(* Logix 5000 project; controller cal1615 1756-L62 rev 20.19; software revision 20.05; part 2 of 82 *)

TYPE Accumulator :
STRUCT
   OUT_Not_EStop : BOOL;   // E-Stop Not Requested
   OUT_Not_Fast_Stop : BOOL;   // Fast Stop Not Requested
   OUT_Not_Normal_Stop : BOOL;   // Normal Stop Not Requested
   OUT_Request_Line_Slowdown : BOOL;   // Request Line Slowdown
   OUT_Full : BOOL;   // Accumulator is Full
   OUT_Empty : BOOL;   // Accumulator is Empty
   OUT_Alarm : BOOL;   // Alarm Exists
   OUT_Unack_Alarm : BOOL;   // Unacknowledged Alarm Exists
   OUT_Warning : BOOL;   // Warning Exists
   OUT_Unack_Warning : BOOL;   // Unacknowledged Warning Exists
   OUT_control_limit : BOOL;   // Control Limit Position
   OUT_Speed : REAL;   // Output Speed
   OUT_Nip_Close : BOOL;   // Nip Close Request
   IN_Speed : REAL;   // Input Speed
   OUT_Acc_Payout : BOOL;   // Accumulator Payout
   OUT_Close_Nip : BOOL;   // Close Nip
   OUT_Acc_Fill_Request : BOOL;   // Accumulator Fill Request
END_STRUCT
END_TYPE

TYPE acs800_di_normal :
STRUCT
   faulted : BOOL;
   warning : BOOL;
   running_fwd : BOOL;
   running_rev : BOOL;
   ready : BOOL;
   ctrl_from_net : BOOL;
   ref_from_net : BOOL;
   at_reference : BOOL;
END_STRUCT
END_TYPE

TYPE acs800_do_normal :
STRUCT
   forward : BOOL;
   reverse : BOOL;
   fault_reset : BOOL;
   net_control : BOOL;
   net_reference : BOOL;
END_STRUCT
END_TYPE

TYPE hmi_dint :
STRUCT
   hmi : DINT[16];
   global : DINT[16];
   zone_1 : DINT[16];
   zone_2 : DINT[16];
   zone_3 : DINT[16];
   letoff : DINT[16];
   ts1 : DINT[16];
   ts2 : DINT[16];
   upl : DINT[16];
   lpl : DINT[16];
   wdr : DINT[16];
   wdt : DINT[16];
   splice : DINT[16];
   mrc : DINT[16];
   static : DINT[16];
   imp : DINT[16];
   misc : DINT[16];
   edg : DINT[16];
   slt : DINT[16];
   impreg : DINT[16];
   adv_cooling : DINT[16];
   retraction : DINT[16];
END_STRUCT
END_TYPE

TYPE hmi_real :
STRUCT
   hmi : REAL[112];
   global : REAL[112];
   zone_1 : REAL[112];
   zone_2 : REAL[112];
   zone_3 : REAL[112];
   letoff : REAL[112];
   ts1 : REAL[112];
   ts2 : REAL[112];
   upl : REAL[112];
   lpl : REAL[112];
   wdr : REAL[112];
   wdt : REAL[112];
   splice : REAL[112];
   mrc : REAL[112];
   static : REAL[112];
   impreg : REAL[112];
   misc : REAL[112];
   edg : REAL[112];
   slt : REAL[112];
   adv_cooling : REAL[112];
END_STRUCT
END_TYPE

TYPE PIDE :   // PIDE
STRUCT
   pide_ctrl : PID_ENHANCED;   // Control PID
   pide_autotune : PIDE_AUTOTUNE;   // PID Autotune Data
   ao_cv : REAL;   // Analog Output: Temperature Control Valve
   param_cv_min : REAL;   // Control Valve Minimum Output
   param_cv_max : REAL;   // Control Valve Maximum Output
   param_pv_min : REAL;   // PV Minimum
   param_pv_max : REAL;   // PV Maximum
   pid_manual_sp : REAL;   // Manual Mode Control Valve Setpoint
   pid_ctrl_cv : REAL;   // Control Valve Output
   pid_ctrl_pv : REAL;   // Control Process Variable
   pid_ctrl_sp : REAL;   // Control Setpoint
   pid_ctrl_sp_error : REAL;   // Control Absolute Error
   pid_ctrl_sp_last : REAL;   // Control Setpoint Last Scan
   oneshot : DINT;   // One Shot
   status : DINT;   // Run Status
   enable_deviation_alarm : BOOL;   // Enable Temperature Deviation Alarm
   pb_cv_manual : BOOL;   // Manual Mode Pushbutton
   pb_cv_auto : BOOL;   // Auto Mode Pushbutton
   pid_manual_mode : BOOL;   // Manual Mode
   request_pid_control : BOOL;   // PID Control Request
   request_manual : BOOL;   // PID Manual Mode Request
END_STRUCT
END_TYPE

TYPE recipe :
STRUCT
   name : STRING;
   comments : STRING;
   master_line_speed : REAL;
   zone_1 : zone;
   zone_2 : zone;
   zone_3 : zone;
   line_speed_sp : REAL;
   letoff_tension_sp : REAL;
   acc_tension_sp : REAL;
   acc_fill_pressure_sp : REAL;
   acc_counter_pressure_sp : REAL;
   cure_time_sp : REAL;
   platen_temp_sp : REAL;
   impreg_gap_sp : REAL;
   impreg_gap_ds_offset_sp : REAL;
   impreg_gap_os_offset_sp : REAL;
   impreg_supply_speed_sp : REAL;
   impreg_roll_speed_sp : REAL;
   ts1_mode_sp : REAL;
   ts1_tension_sp : REAL;
   ts1_stretch_sp : REAL;
   liner_winder_brake_sp : REAL;
   slitter_speed_sp : REAL;
   adv_cooling_temp_sp : REAL;
   ts2_tension_sp : REAL;
   lower_poly_tension_sp : REAL;
   lower_poly_b_tension_sp : REAL;
   upper_poly_tension_sp : REAL;
   upper_poly_b_tension_sp : REAL;
   winder_tension_sp : REAL;
   winder_mode_sp : REAL;
   winder_torque_sp : REAL;
   tension_deviation_sp : REAL;
   winder_tension_sp_max : REAL;
   winder_tension_sp_min : REAL;
END_STRUCT
END_TYPE

TYPE routine :
STRUCT
   comment : DINT;
   oneshot : DINT;
   fault : DINT;
   fault_ack : DINT;
   fault1 : DINT;
   fault1_ack : DINT;
   warning : DINT;
   warning_ack : DINT;
   unack_fault : BOOL;
   unack_warning : BOOL;
   state : DINT;
END_STRUCT
END_TYPE

TYPE servo_di :
STRUCT
   mode_bit_0 : BOOL;
   mode_bit_1 : BOOL;
   homed : BOOL;
   stand_still : BOOL;
   at_target_pos : BOOL;
   command_change : BOOL;
   operator_mode_error : BOOL;
   drive_does_not_follow : BOOL;
   actual_op_mode_bit_0 : BOOL;
   actual_op_mode_bit_1 : BOOL;
   class_3_diagnostic : BOOL;
   class_2_diagnostic : BOOL;
   class_1_diagnostic : BOOL;
   operation_bit_14 : BOOL;
   operation_bit_15 : BOOL;
END_STRUCT
END_TYPE

TYPE servo_do :
STRUCT
   command_value_accept : BOOL;
   fault_reset : BOOL;
   jog_forward : BOOL;
   jog_reverse : BOOL;
   jog_enable : BOOL;
   drive_halt_0_halt : BOOL;
   drive_enable : BOOL;
   ready_for_operation_bit_16 : BOOL;
   ready_for_operation_bit_17 : BOOL;
END_STRUCT
END_TYPE

TYPE Setpoint :   // ******************** DO NOT CHANGE ORDER OF TAGS ******************** ****
STRUCT
   SP : REAL;   // Setpoint
   Lo : REAL;   // Lo
   Hi : REAL;   // Hi
END_STRUCT
END_TYPE

TYPE vfd_data :
STRUCT
   In_OutputFreq : DINT;
   In_RPM : DINT;
   In_OutputCurrent : DINT;
   In_MaximumFreq : DINT;
   In_MotorNPHz : DINT;
   In_MotorNPRPM : DINT;
   In_DriveStatus : DINT;
   Out_CommandedFreq : DINT;
   Out_DriveLogicRslt : DINT;
   Out_CommandedRPM : DINT;
   In_DriveStatus_Ready : BOOL;
   In_DriveStatus_Active : BOOL;
   In_DriveStatus_Faulted : BOOL;
   In_DriveStatus_Net : BOOL;
   In_DriveStatus_AtReference : BOOL;
   Out_DriveLogicRslt_Stop : BOOL;
   Out_DriveLogicRslt_Start : BOOL;
   Out_DriveLogicRslt_ClearFault : BOOL;
   Out_DriveLogicRslt_Forward : BOOL;
   Out_DriveLogicRslt_Reverse : BOOL;
END_STRUCT
END_TYPE

TYPE vfd_data_ACS880 :
STRUCT
   In_OutputRPM : DINT;   // Input
   In_OutputCurrent : DINT;   // Input
   IN_OutputHz : DINT;   // Output Hz
   IN_OutputTorque : DINT;   // Input Motor Torque
   In_SpeedScaling : DINT;   // Input
   In_MotorNPHz : DINT;   // Input
   In_MotorNPRPM : DINT;   // Input
   In_DriveStatus : DINT;   // Input
   Out_DriveLogicRslt : DINT;   // Output
   Out_Speed_Setpoint : REAL;   // Motor Speed Setpoint in Engineering Units
   Out_SpeedScaling : DINT;   // Output Speed Scaling
   Out_Commanded_SPEED : REAL;   // Output
   Out_Commanded_Torque : REAL;   // Output Torque
   C_speed_hz : BOOL;   // Speed Setpoint in Hz
   C_speed_pct : BOOL;   // Speed Setpoint In Percent
   C_speed_rpm : BOOL;   // Speed Setpoint in RPM
   In_DriveStatus_RDY_ON : BOOL;   // Input
   In_DriveStatus_RDY_RUN : BOOL;   // Input
   In_DriveStatus_RDY_REF : BOOL;   // Input
   In_DriveStatus_TRIPPED : BOOL;   // Input Status Tripped
   In_DriveStatus_OFF_2_STA : BOOL;   // Input Status Off 2 State
   In_DriveStatus_OFF_3_STA : BOOL;   // Input Status Off 3 State
   In_DriveStatus_SWC_ON_INHIB : BOOL;   // Input Status SWC On Inhibit
   In_DriveStatus_ALARM : BOOL;   // Input Status Alarm
   In_DriveStatus_AT_SETPOINT : BOOL;   // Input Status At Setpoint
   In_DriveStatus_REMOTE : BOOL;   // Input Status Remote
   In_DriveStatus_ABOVE_LIMIT : BOOL;   // Input Status Above Limit
   In_DriveStatus_EXT_CTRL_LOC : BOOL;   // Input Status External Control
   In_DriveStatus_EXT_RUN_ENABLE : BOOL;   // Input Status External Run Enable
   In_DriveStatus_FBA_ERROR : BOOL;   // Input Status Field Bus Error
   Out_DriveLogicRslt_OFF1_CONTROL : BOOL;   // Output Off 1 Control
   Out_DriveLogicRslt_OFF2_CONTROL : BOOL;   // Output Off 2 Control
   Out_DriveLogicRslt_OFF3_CONTROL : BOOL;   // Output Off 3 Control
   Out_DriveLogicRslt_INHIBIT_OPERATION : BOOL;   // Output Inhibit Operation
   Out_DriveLogicRslt_RAMP_OUT_ZERO : BOOL;   // Output Ramp Out Zero
   Out_DriveLogicRslt_RAMP_HOLD : BOOL;   // Output Ramp Hold
   Out_DriveLogicRslt_RAMP_IN_ZERO : BOOL;   // Output Ramp In Zero
   Out_DriveLogicRslt_RESET : BOOL;   // Output Reset
   Out_DriveLogicRslt_REMOTE_CMD : BOOL;   // Output Remmote Command
   Out_DriveLogicRslt_EXT_CTRL_LOC : BOOL;   // Output Ext Ctrl Loc
   OUT_Comm_Status : BOOL;
END_STRUCT
END_TYPE

TYPE zone :
STRUCT
   recirc_sp : REAL;
   exhaust_sp : REAL;
   temp_sp : REAL;
END_STRUCT
END_TYPE

ADD_ON_INSTRUCTION ABB_PROTOCOL_VFD   (* revision 1.0 *)
VAR_INPUT
   STATUS_WORD : INT; {required}
END_VAR
VAR_OUTPUT
   CONTROL_WORD : INT; {access Read Only, required}
END_VAR
VAR_INPUT
   DRIVE_NOT_READY_FAULT : BOOL;
END_VAR
VAR_OUTPUT
   OUT_FAULT : BOOL; {access Read Only, visible}
   OUT_ALARM : BOOL; {access Read Only, visible}
   OUT_ENABLED : BOOL; {access Read Only, visible}
END_VAR
VAR_INPUT
   IN_START : BOOL; {required}
   IN_GLOBAL_RESET : BOOL; {required}
   IN_DRIVE_PERMISSIVE : BOOL; {required}
END_VAR
VAR
   run_permissive : BOOL;
   enable_drives : BOOL;
   request_run : BOOL;
   drive_on_request : BOOL;
   seq : routine;
   step_3_timer : TIMER := (PRE := 500);
   fault_timer : TIMER := (PRE := 2000);
END_VAR

ROUTINE Logic   (* ladder *)
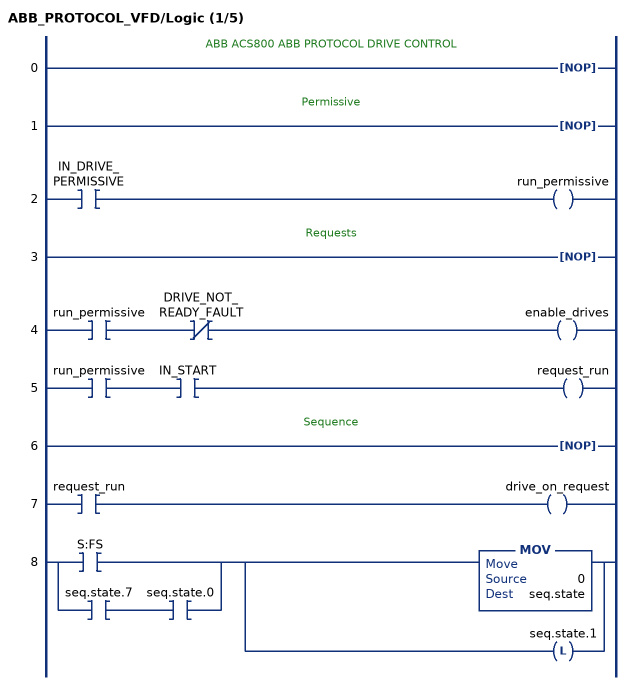
   // ABB ACS800 ABB PROTOCOL DRIVE CONTROL
   0: NOP();
   // Permissive
   1: NOP();
   2: XIC(IN_DRIVE_PERMISSIVE)OTE(run_permissive);
   // Requests
   3: NOP();
   4: XIC(run_permissive)XIO(DRIVE_NOT_READY_FAULT)OTE(enable_drives);
   5: XIC(run_permissive)XIC(IN_START)OTE(request_run);
   // Sequence
   6: NOP();
   7: XIC(request_run)OTE(drive_on_request);
   8: [XIC(S:FS) ,XIC(seq.state.7) XIC(seq.state.0) ][MOV(0,seq.state) ,OTL(seq.state.1) ];
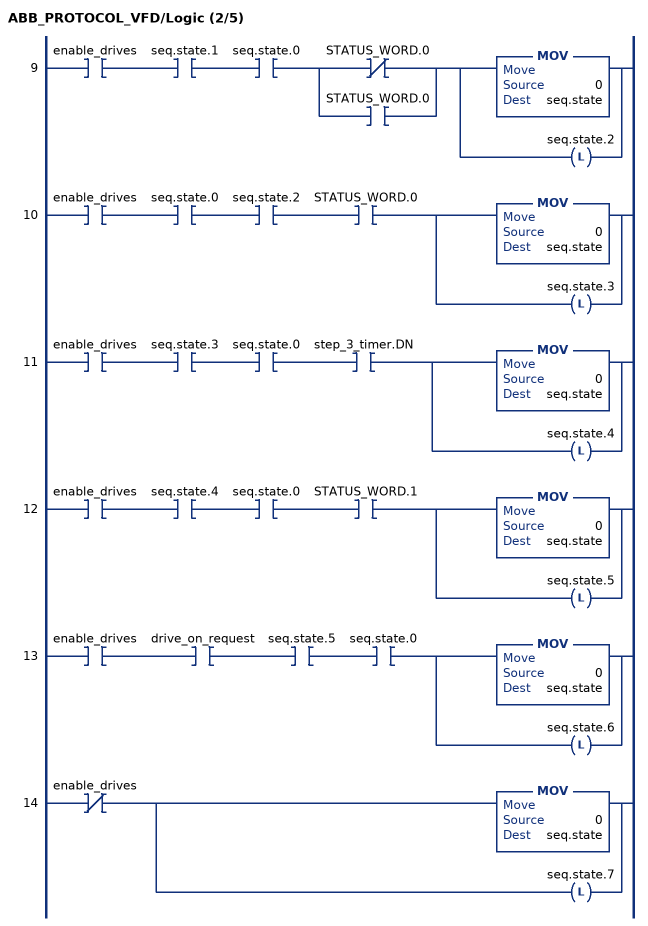
   9: XIC(enable_drives)XIC(seq.state.1)XIC(seq.state.0)[XIO(STATUS_WORD.0) ,XIC(STATUS_WORD.0) ][MOV(0,seq.state) ,OTL(seq.state.2) ];
   10: XIC(enable_drives)XIC(seq.state.0)XIC(seq.state.2)XIC(STATUS_WORD.0)[MOV(0,seq.state) ,OTL(seq.state.3) ];
   11: XIC(enable_drives)XIC(seq.state.3)XIC(seq.state.0)XIC(step_3_timer.DN)[MOV(0,seq.state) ,OTL(seq.state.4) ];
   12: XIC(enable_drives)XIC(seq.state.4)XIC(seq.state.0)XIC(STATUS_WORD.1)[MOV(0,seq.state) ,OTL(seq.state.5) ];
   13: XIC(enable_drives)XIC(drive_on_request)XIC(seq.state.5)XIC(seq.state.0)[MOV(0,seq.state) ,OTL(seq.state.6) ];
   14: XIO(enable_drives)[MOV(0,seq.state) ,OTL(seq.state.7) ];
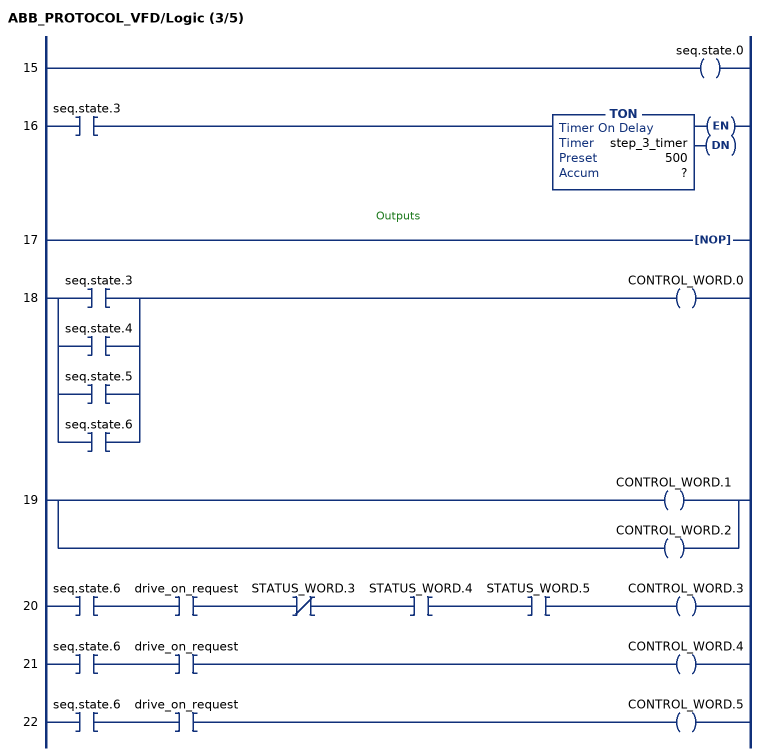
   15: OTE(seq.state.0);
   16: XIC(seq.state.3)TON(step_3_timer,?,?);
   // Outputs
   17: NOP();
   18: [XIC(seq.state.3) ,XIC(seq.state.4) ,XIC(seq.state.5) ,XIC(seq.state.6) ]OTE(CONTROL_WORD.0);
   19: [OTE(CONTROL_WORD.1) ,OTE(CONTROL_WORD.2) ];
   20: XIC(seq.state.6)XIC(drive_on_request)XIO(STATUS_WORD.3)XIC(STATUS_WORD.4)XIC(STATUS_WORD.5)OTE(CONTROL_WORD.3);
   21: XIC(seq.state.6)XIC(drive_on_request)OTE(CONTROL_WORD.4);
   22: XIC(seq.state.6)XIC(drive_on_request)OTE(CONTROL_WORD.5);
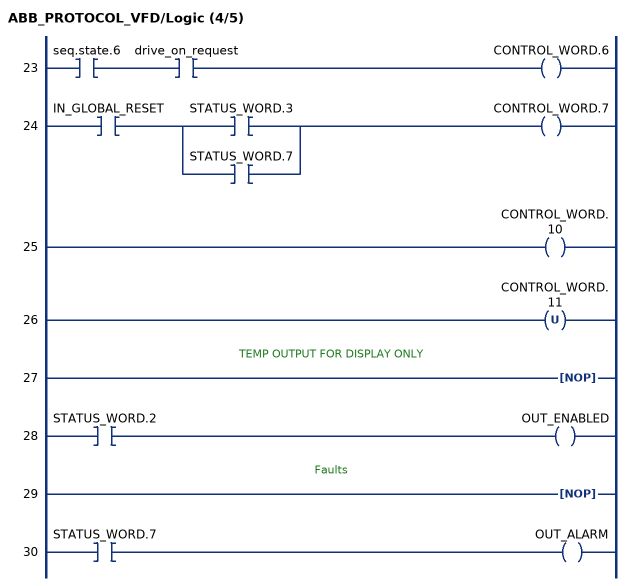
   23: XIC(seq.state.6)XIC(drive_on_request)OTE(CONTROL_WORD.6);
   24: XIC(IN_GLOBAL_RESET)[XIC(STATUS_WORD.3) ,XIC(STATUS_WORD.7) ]OTE(CONTROL_WORD.7);
   25: OTE(CONTROL_WORD.10);
   26: OTU(CONTROL_WORD.11);
   // TEMP OUTPUT FOR DISPLAY ONLY
   27: NOP();
   28: XIC(STATUS_WORD.2)OTE(OUT_ENABLED);
   // Faults
   29: NOP();
   30: XIC(STATUS_WORD.7)OTE(OUT_ALARM);
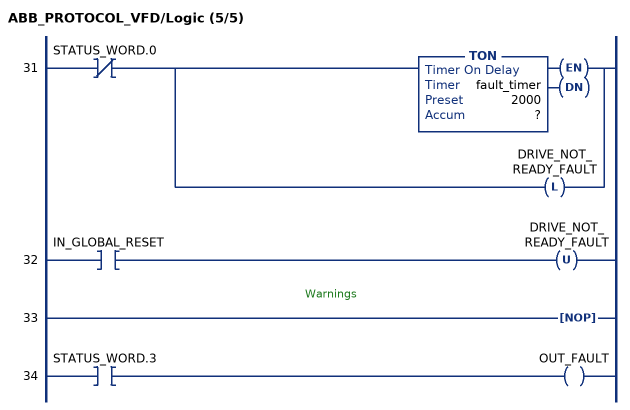
   31: XIO(STATUS_WORD.0)[TON(fault_timer,?,?) ,OTL(DRIVE_NOT_READY_FAULT) ];
   32: XIC(IN_GLOBAL_RESET)OTU(DRIVE_NOT_READY_FAULT);
   // Warnings
   33: NOP();
   34: XIC(STATUS_WORD.3)OTE(OUT_FAULT);
END_ROUTINE
END_ADD_ON_INSTRUCTION

ADD_ON_INSTRUCTION ARM_PID   (* revision 1.0 *)
VAR_IN_OUT
   PID : PID; {required}   // PID
END_VAR
VAR_INPUT
   NOBC : BOOL; {required}   // No Bias Calculation
   CA : BOOL; {required}   // Control
   Min : REAL; {required}   // Min (Scale/Eng)
   Max : REAL; {required}   // Max (Scale/Eng)
END_VAR

ROUTINE Logic   (* ladder *)
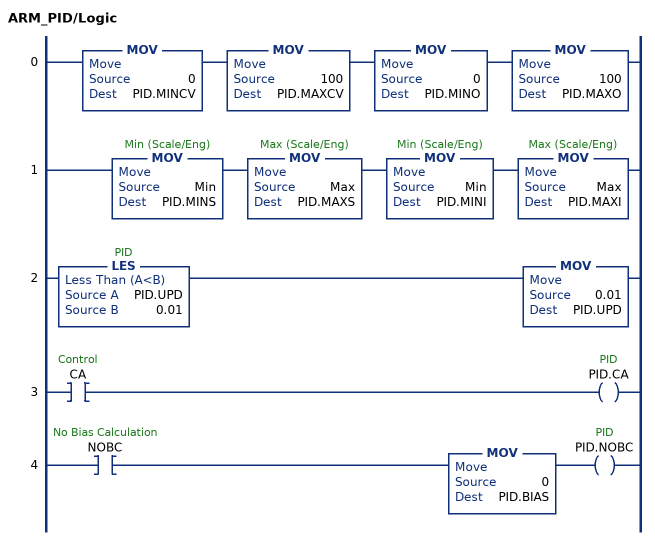
   0: MOV(0,PID.MINCV)MOV(100,PID.MAXCV)MOV(0,PID.MINO)MOV(100,PID.MAXO);
   1: MOV(Min,PID.MINS)MOV(Max,PID.MAXS)MOV(Min,PID.MINI)MOV(Max,PID.MAXI);
   2: LES(PID.UPD,0.01)MOV(0.01,PID.UPD);
   3: XIC(CA)OTE(PID.CA);
   4: XIC(NOBC)MOV(0,PID.BIAS)OTE(PID.NOBC);
END_ROUTINE
END_ADD_ON_INSTRUCTION

ADD_ON_INSTRUCTION Limit_Clamp   (* revision 1.0 *)
VAR_INPUT
   max : REAL; {required}
END_VAR
VAR_IN_OUT
   variable : REAL; {required}
END_VAR
VAR_INPUT
   min : REAL; {required}
END_VAR

ROUTINE Logic   (* ladder *)
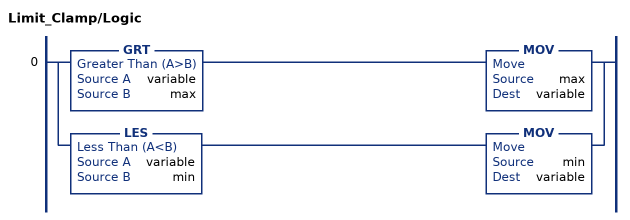
   0: [GRT(variable,max) MOV(max,variable) ,LES(variable,min) MOV(min,variable) ];
END_ROUTINE
END_ADD_ON_INSTRUCTION

ADD_ON_INSTRUCTION Ramp_Test   (* revision 1.0 *)
VAR_INPUT
   SP : REAL; {required}
   Rate : REAL; {required}
   ScanTime : REAL; {required}
END_VAR
VAR_IN_OUT
   PV : REAL; {required}
END_VAR
VAR
   request_decel : BOOL;
   request_accel : BOOL;
END_VAR

ROUTINE Logic   (* ladder *)
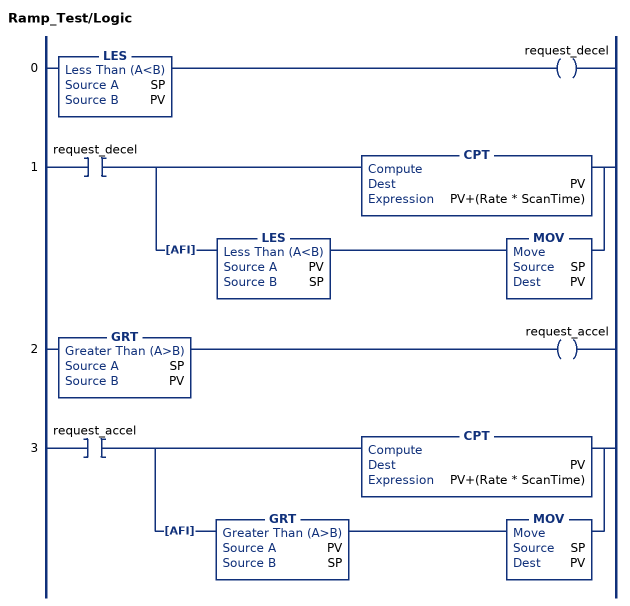
   0: LES(SP,PV)OTE(request_decel);
   1: XIC(request_decel)[CPT(PV,PV+(Rate * ScanTime)) ,AFI() LES(PV,SP) MOV(SP,PV) ];
   2: GRT(SP,PV)OTE(request_accel);
   3: XIC(request_accel)[CPT(PV,PV+(Rate * ScanTime)) ,AFI() GRT(PV,SP) MOV(SP,PV) ];
END_ROUTINE
END_ADD_ON_INSTRUCTION

ADD_ON_INSTRUCTION SYS_ACC_DEC_RAMP   (* revision 1.0 *)
VAR_INPUT
   IN_selected_line_speed : REAL; {required}   // Input Parameter Selected Line Speed
   IN_param_master_accel_rate : REAL; {required}   // Input Parameter Acel Ramp x/second
   IN_param_master_decel_rate : REAL; {required}   // Input Parameter Decel Ramp x/second
   IN_last_scan_s : REAL; {required}   // Input Parameter Last Scan seconds
END_VAR
VAR_IN_OUT
   IN_OUT_master_ramped_speed : REAL; {required}   // Input Output Parameter Master Ramped Speed
END_VAR
VAR
   p01r03_last_scan_ms : DINT;
   local_last_scan_ms : DINT;
END_VAR

ROUTINE Logic   (* ladder *)
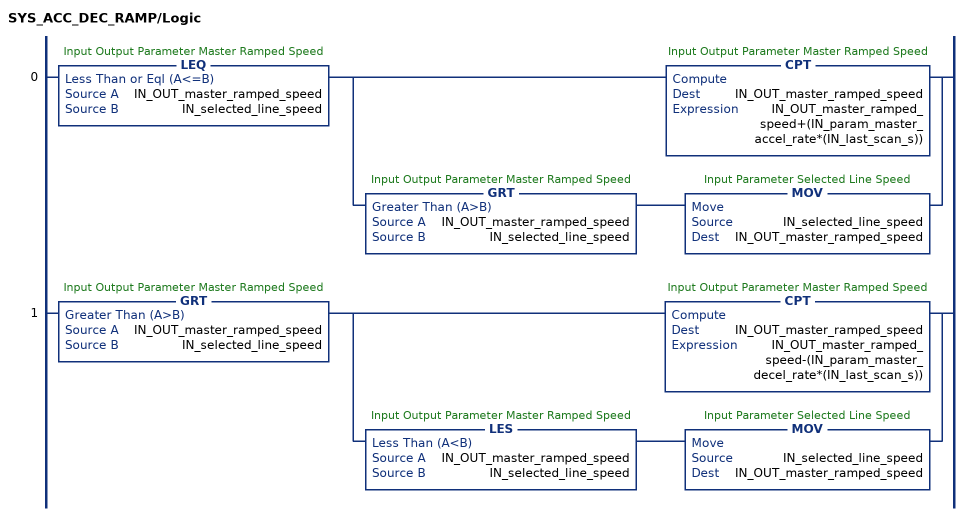
   0: LEQ(IN_OUT_master_ramped_speed,IN_selected_line_speed)[CPT(IN_OUT_master_ramped_speed,IN_OUT_master_ramped_speed+(IN_param_master_accel_rate*(IN_last_scan_s))) ,GRT(IN_OUT_master_ramped_speed,IN_selected_line_speed) MOV(IN_selected_line_speed,IN_OUT_master_ramped_speed) ];
   1: GRT(IN_OUT_master_ramped_speed,IN_selected_line_speed)[CPT(IN_OUT_master_ramped_speed,IN_OUT_master_ramped_speed-(IN_param_master_decel_rate*(IN_last_scan_s))) ,LES(IN_OUT_master_ramped_speed,IN_selected_line_speed) MOV(IN_selected_line_speed,IN_OUT_master_ramped_speed) ];
END_ROUTINE
END_ADD_ON_INSTRUCTION

ADD_ON_INSTRUCTION sys_Acknowledge   (* revision 1.0, vendor Rockwell Automation *)
VAR_IN_OUT
   Ack : DINT; {required}
END_VAR
VAR_INPUT
   Alarm : DINT; {required}
END_VAR

ROUTINE Logic   (* ladder *)
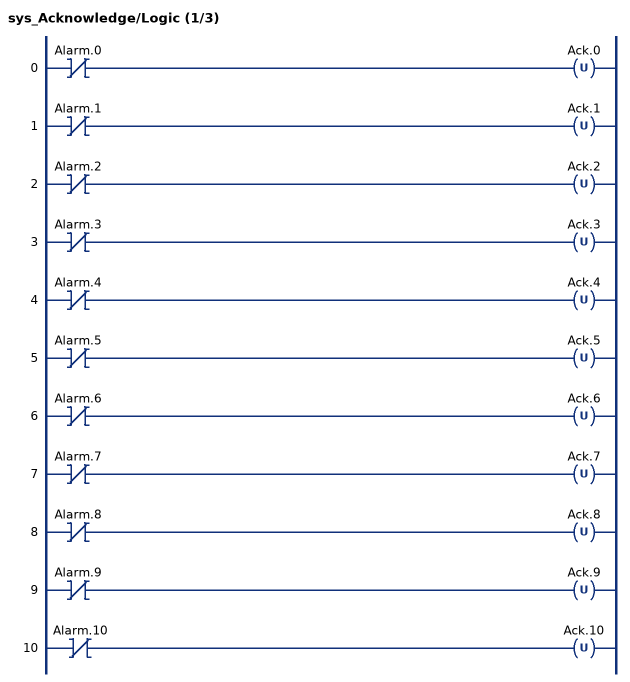
   0: XIO(Alarm.0)OTU(Ack.0);
   1: XIO(Alarm.1)OTU(Ack.1);
   2: XIO(Alarm.2)OTU(Ack.2);
   3: XIO(Alarm.3)OTU(Ack.3);
   4: XIO(Alarm.4)OTU(Ack.4);
   5: XIO(Alarm.5)OTU(Ack.5);
   6: XIO(Alarm.6)OTU(Ack.6);
   7: XIO(Alarm.7)OTU(Ack.7);
   8: XIO(Alarm.8)OTU(Ack.8);
   9: XIO(Alarm.9)OTU(Ack.9);
   10: XIO(Alarm.10)OTU(Ack.10);
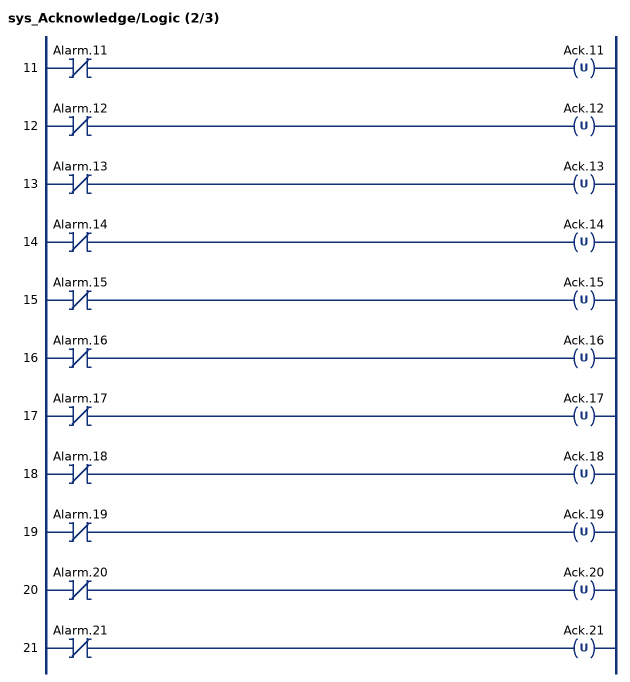
   11: XIO(Alarm.11)OTU(Ack.11);
   12: XIO(Alarm.12)OTU(Ack.12);
   13: XIO(Alarm.13)OTU(Ack.13);
   14: XIO(Alarm.14)OTU(Ack.14);
   15: XIO(Alarm.15)OTU(Ack.15);
   16: XIO(Alarm.16)OTU(Ack.16);
   17: XIO(Alarm.17)OTU(Ack.17);
   18: XIO(Alarm.18)OTU(Ack.18);
   19: XIO(Alarm.19)OTU(Ack.19);
   20: XIO(Alarm.20)OTU(Ack.20);
   21: XIO(Alarm.21)OTU(Ack.21);
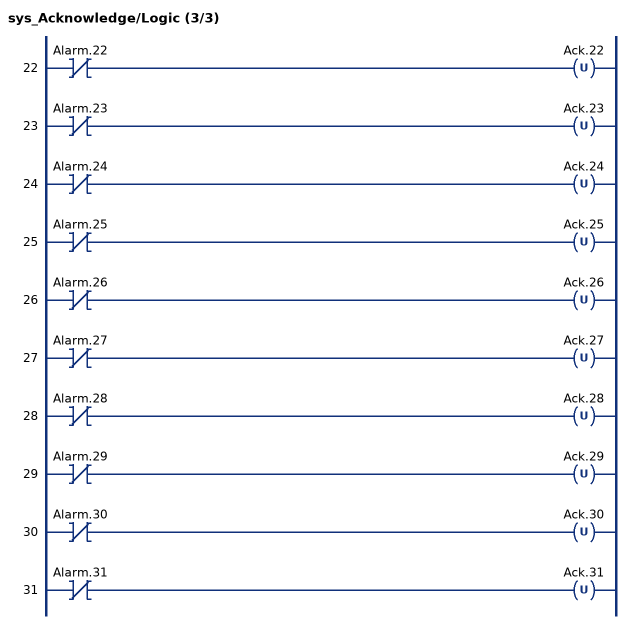
   22: XIO(Alarm.22)OTU(Ack.22);
   23: XIO(Alarm.23)OTU(Ack.23);
   24: XIO(Alarm.24)OTU(Ack.24);
   25: XIO(Alarm.25)OTU(Ack.25);
   26: XIO(Alarm.26)OTU(Ack.26);
   27: XIO(Alarm.27)OTU(Ack.27);
   28: XIO(Alarm.28)OTU(Ack.28);
   29: XIO(Alarm.29)OTU(Ack.29);
   30: XIO(Alarm.30)OTU(Ack.30);
   31: XIO(Alarm.31)OTU(Ack.31);
END_ROUTINE
END_ADD_ON_INSTRUCTION

ADD_ON_INSTRUCTION sys_ACS880_inputs   (* revision 1.0 *)
// System AOI
// ACS880 Inputs
VAR_IN_OUT
   IN_vfd_inputs : AB:ETHERNET_MODULE_INT_24Bytes:I:0; {required}
   IN_vfd_data : vfd_data_ACS880; {required}
END_VAR
VAR_INPUT
   IN_vfd_status : DINT; {required}
END_VAR
VAR_OUTPUT
   Out_RPM : REAL; {access Read Only, required}
   Out_Amps : REAL; {access Read Only, required}
   Out_Hz : REAL; {access Read Only, required}
   Out_TorquePct : REAL; {access Read Only, required}
   Out_Speed : REAL; {access Read Only, required}
END_VAR
VAR_INPUT
   IN_Roll_Diameter : REAL; {required}
   IN_Gear_Reduction : REAL; {required}
END_VAR
VAR
   afi : BOOL;
   comm_ok : BOOL;
   NPRPM : DINT;
   NPHz : DINT;
END_VAR

ROUTINE Logic   (* ladder *)
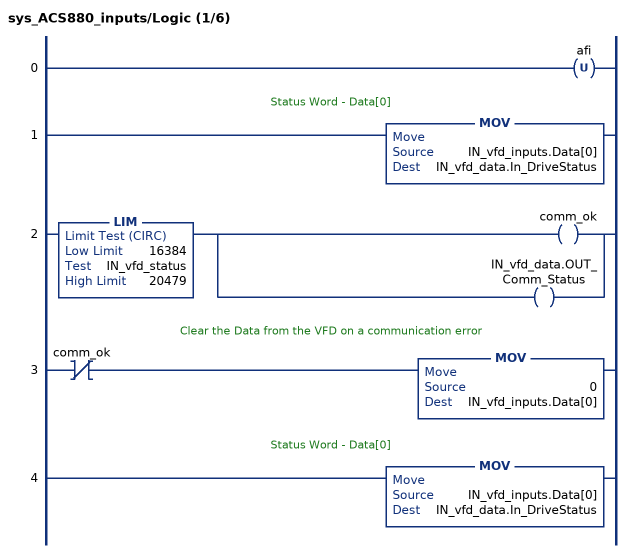
   0: OTU(afi);
   // Status Word - Data[0]
   1: MOV(IN_vfd_inputs.Data[0],IN_vfd_data.In_DriveStatus);
   2: LIM(16384,IN_vfd_status,20479)[OTE(comm_ok) ,OTE(IN_vfd_data.OUT_Comm_Status) ];
   // Clear the Data from the VFD on a communication error
   3: XIO(comm_ok)MOV(0,IN_vfd_inputs.Data[0]);
   // Status Word - Data[0]
   4: MOV(IN_vfd_inputs.Data[0],IN_vfd_data.In_DriveStatus);
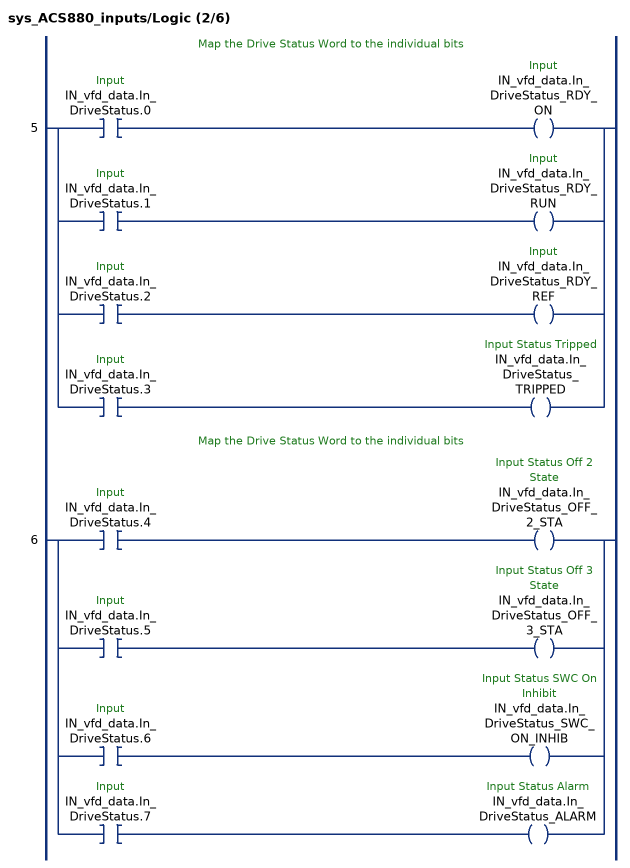
   // Map the Drive Status Word to the individual bits
   5: [XIC(IN_vfd_data.In_DriveStatus.0) OTE(IN_vfd_data.In_DriveStatus_RDY_ON) ,XIC(IN_vfd_data.In_DriveStatus.1) OTE(IN_vfd_data.In_DriveStatus_RDY_RUN) ,XIC(IN_vfd_data.In_DriveStatus.2) OTE(IN_vfd_data.In_DriveStatus_RDY_REF) ,XIC(IN_vfd_data.In_DriveStatus.3) OTE(IN_vfd_data.In_DriveStatus_TRIPPED) ];
   // Map the Drive Status Word to the individual bits
   6: [XIC(IN_vfd_data.In_DriveStatus.4) OTE(IN_vfd_data.In_DriveStatus_OFF_2_STA) ,XIC(IN_vfd_data.In_DriveStatus.5) OTE(IN_vfd_data.In_DriveStatus_OFF_3_STA) ,XIC(IN_vfd_data.In_DriveStatus.6) OTE(IN_vfd_data.In_DriveStatus_SWC_ON_INHIB) ,XIC(IN_vfd_data.In_DriveStatus.7) OTE(IN_vfd_data.In_DriveStatus_ALARM) ];
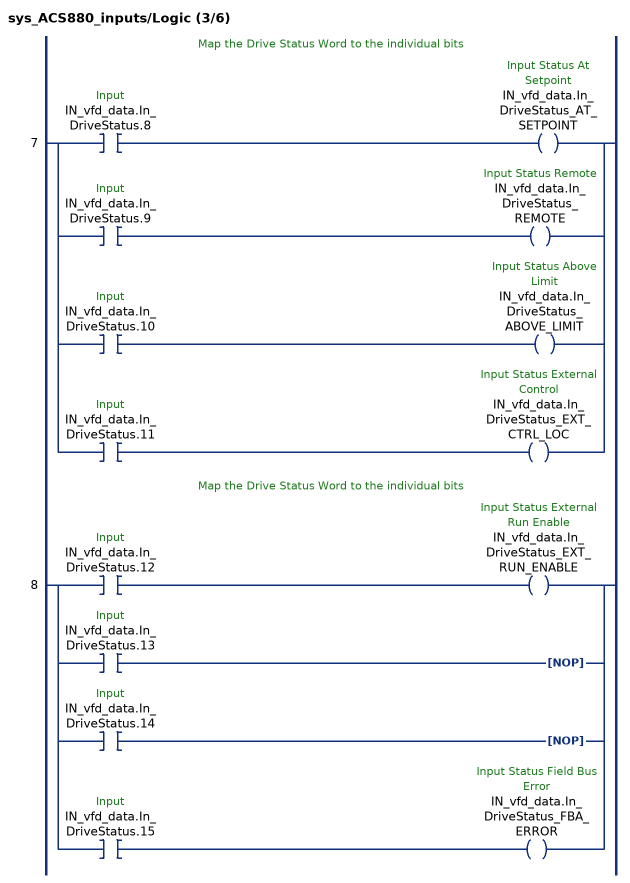
   // Map the Drive Status Word to the individual bits
   7: [XIC(IN_vfd_data.In_DriveStatus.8) OTE(IN_vfd_data.In_DriveStatus_AT_SETPOINT) ,XIC(IN_vfd_data.In_DriveStatus.9) OTE(IN_vfd_data.In_DriveStatus_REMOTE) ,XIC(IN_vfd_data.In_DriveStatus.10) OTE(IN_vfd_data.In_DriveStatus_ABOVE_LIMIT) ,XIC(IN_vfd_data.In_DriveStatus.11) OTE(IN_vfd_data.In_DriveStatus_EXT_CTRL_LOC) ];
   // Map the Drive Status Word to the individual bits
   8: [XIC(IN_vfd_data.In_DriveStatus.12) OTE(IN_vfd_data.In_DriveStatus_EXT_RUN_ENABLE) ,XIC(IN_vfd_data.In_DriveStatus.13) NOP() ,XIC(IN_vfd_data.In_DriveStatus.14) NOP() ,XIC(IN_vfd_data.In_DriveStatus.15) OTE(IN_vfd_data.In_DriveStatus_FBA_ERROR) ];
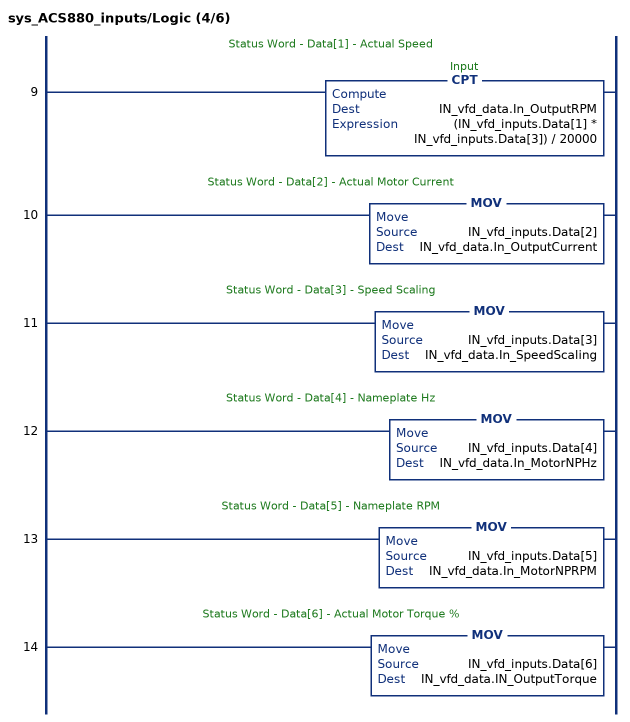
   // Status Word - Data[1] - Actual Speed
   9: CPT(IN_vfd_data.In_OutputRPM,(IN_vfd_inputs.Data[1] * IN_vfd_inputs.Data[3]) / 20000);
   // Status Word - Data[2] - Actual Motor Current
   10: MOV(IN_vfd_inputs.Data[2],IN_vfd_data.In_OutputCurrent);
   // Status Word - Data[3] - Speed Scaling
   11: MOV(IN_vfd_inputs.Data[3],IN_vfd_data.In_SpeedScaling);
   // Status Word - Data[4] - Nameplate Hz
   12: MOV(IN_vfd_inputs.Data[4],IN_vfd_data.In_MotorNPHz);
   // Status Word - Data[5] - Nameplate RPM
   13: MOV(IN_vfd_inputs.Data[5],IN_vfd_data.In_MotorNPRPM);
   // Status Word - Data[6] - Actual Motor Torque %
   14: MOV(IN_vfd_inputs.Data[6],IN_vfd_data.IN_OutputTorque);
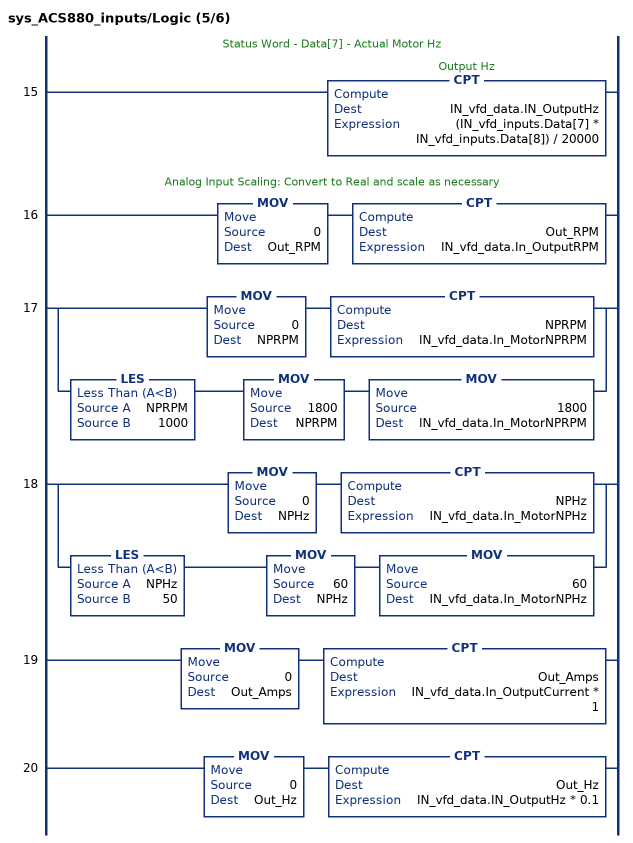
   // Status Word - Data[7] - Actual Motor Hz
   15: CPT(IN_vfd_data.IN_OutputHz,(IN_vfd_inputs.Data[7] * IN_vfd_inputs.Data[8]) / 20000);
   // Analog Input Scaling: Convert to Real and scale as necessary
   16: MOV(0,Out_RPM)CPT(Out_RPM,IN_vfd_data.In_OutputRPM);
   17: [MOV(0,NPRPM) CPT(NPRPM,IN_vfd_data.In_MotorNPRPM) ,LES(NPRPM,1000) MOV(1800,NPRPM) MOV(1800,IN_vfd_data.In_MotorNPRPM) ];
   18: [MOV(0,NPHz) CPT(NPHz,IN_vfd_data.In_MotorNPHz) ,LES(NPHz,50) MOV(60,NPHz) MOV(60,IN_vfd_data.In_MotorNPHz) ];
   19: MOV(0,Out_Amps)CPT(Out_Amps,IN_vfd_data.In_OutputCurrent * 1);
   20: MOV(0,Out_Hz)CPT(Out_Hz,IN_vfd_data.IN_OutputHz * 0.1);
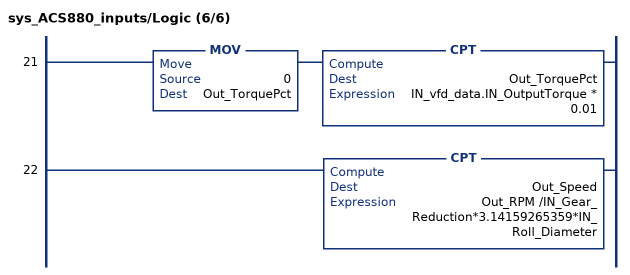
   21: MOV(0,Out_TorquePct)CPT(Out_TorquePct,IN_vfd_data.IN_OutputTorque * 0.01);
   22: CPT(Out_Speed,Out_RPM /IN_Gear_Reduction*3.14159265359*IN_Roll_Diameter);
END_ROUTINE
END_ADD_ON_INSTRUCTION
